Staubli VAL3: setConveyor.pgx

public program setConveyor(frame& x_fFrame)
begin
  // This programs sets the input frame as conveyor
  //
  // Input Param
  //  x_fFrame   : Frame to be set as conveyor
  //
  // Output Param
  //  none       :
  //
  //----------------------------------------------------------------
  //
  // The frame may be already conveyor (previous run)
  $setMobile(x_fFrame,false)
  // Set frame as conveyor
  $setConv(x_fFrame,enc:aiEncCurrentPos,"pos",{nENCSCALEFACTOR,0,0,0,0,0},nFirTime,nFirDelay)
end
